FUNCTION_BLOCK PauseSwitch
  (* Standard: 61499-2 *)
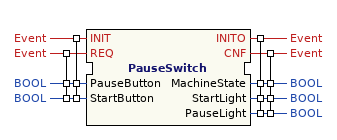
  EVENT_INPUT
    INIT WITH PauseButton, StartButton;
    REQ WITH PauseButton, StartButton;
  END_EVENT
  EVENT_OUTPUT
    INITO WITH MachineState, StartLight, PauseLight;
    CNF WITH MachineState, StartLight, PauseLight;
  END_EVENT
  VAR_INPUT
    PauseButton : BOOL;
    StartButton : BOOL;
  END_VAR
  VAR_OUTPUT
    MachineState : BOOL;
    StartLight : BOOL;
    PauseLight : BOOL;
  END_VAR
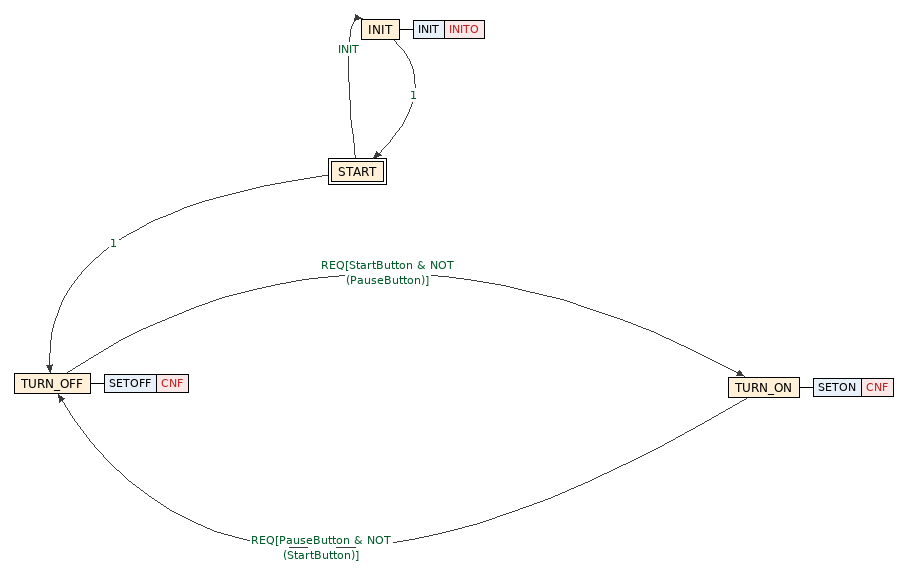
  EC_STATES
    START;
    INIT : INIT -> INITO;
    TURN_ON : SETON -> CNF;
    TURN_OFF : SETOFF -> CNF;
  END_STATES
  EC_TRANSITIONS
    START TO INIT := INIT;
    INIT TO START := 1;
    START TO TURN_OFF := 1;
    TURN_ON TO TURN_OFF := REQ[PauseButton & NOT (StartButton)];
    TURN_OFF TO TURN_ON := REQ[StartButton & NOT (PauseButton)];
  END_TRANSITIONS
  ALGORITHM INIT IN ST:

  END_ALGORITHM
  ALGORITHM SETON IN ST:
MachineState := 1;&#10;StartLight := 1;&#10;PauseLight := 0;&#10;
  END_ALGORITHM
  ALGORITHM SETOFF IN ST:
MachineState := 0;&#10;StartLight := 0;&#10;PauseLight := 1;&#10;
  END_ALGORITHM
END_FUNCTION_BLOCK
